PROGRAM Permissives
VAR
	
	
END_VAR

IF (LCP1_IO.Segment[1].ChargeRly_close = TRUE AND 
	LCP1_IO.Segment[2].ChargeRly_close = TRUE AND
	LCP1_IO.Segment[3].ChargeRly_close = TRUE AND 
	LCP2_IO.Segment[4].ChargeRly_close = TRUE AND 
	LCP2_IO.Segment[5].ChargeRly_close = TRUE AND 
	LCP2_IO.Segment[6].ChargeRly_close = TRUE) OR HMI_DB.AllChargeRelayCloseBP = TRUE
	THEN 
		Permissives_DB.AllChargeRelayClosed := TRUE;
	ELSIF 
		LCP1_IO.Segment[1].ChargeRly_close = FALSE AND 
		LCP1_IO.Segment[2].ChargeRly_close = FALSE AND
		LCP1_IO.Segment[3].ChargeRly_close = FALSE AND 
		LCP2_IO.Segment[4].ChargeRly_close = FALSE AND 
		LCP2_IO.Segment[5].ChargeRly_close = FALSE AND 
		LCP2_IO.Segment[6].ChargeRly_close = FALSE
	THEN
		Permissives_DB.AllChargeRelayClosed := FALSE;
END_IF;

IF (LCP1_IO.Segment[1].Module1To3DumpRly_close = FALSE AND 
	LCP1_IO.Segment[2].Module4To6DumpRly_close = FALSE AND
	LCP1_IO.Segment[3].Module7To9DumpRly_close = FALSE AND
	
	LCP2_IO.Segment[4].Module1To3DumpRly_close = FALSE AND 
	LCP2_IO.Segment[5].Module4To6DumpRly_close = FALSE AND
	LCP2_IO.Segment[6].Module7To9DumpRly_close = FALSE) OR HMI_DB.AllDumpRelaysOpenBP = TRUE
	THEN
		Permissives_DB.AllDumpRelayOpen := TRUE;
		ELSIF
			LCP1_IO.Segment[1].Module1To3DumpRly_close = TRUE AND 
			LCP1_IO.Segment[2].Module4To6DumpRly_close = TRUE AND
			LCP1_IO.Segment[3].Module7To9DumpRly_close = TRUE AND
			LCP2_IO.Segment[4].Module1To3DumpRly_close = TRUE AND
			LCP2_IO.Segment[5].Module4To6DumpRly_close = TRUE AND
			LCP2_IO.Segment[6].Module7To9DumpRly_close = TRUE 
		THEN
			Permissives_DB.AllDumpRelayOpen := FALSE;
END_IF;

IF Permissives_DB.AllChargeRelayClosed = TRUE AND 
	Permissives_DB.AllDumpRelayOpen = TRUE AND
	(Permissives_DB.AllVoltMonBoardStatusOK= TRUE OR HMI_DB.AllVoltMonBoardStatusOKBP = TRUE)  //voltmonitor board has missing packets, so this might be sensitive and might need to bypass
	THEN
		Permissives_DB.ReadyToCharge := TRUE;
	ELSE 
		Permissives_DB.ReadyToCharge := FALSE;
END_IF

IF MCP_IO.Charger[1].voltageFeedback <= Permissives_DB.ChargerVThres AND 
	MCP_IO.Charger[2].voltageFeedback <= Permissives_DB.ChargerVThres AND 
	MCP_IO.Charger[3].voltageFeedback <= Permissives_DB.ChargerVThres AND
	MCP_IO.Charger[4].voltageFeedback <= Permissives_DB.ChargerVThres AND
	MCP_IO.Charger[5].voltageFeedback <= Permissives_DB.ChargerVThres AND
	MCP_IO.Charger[6].voltageFeedback <= Permissives_DB.ChargerVThres
	THEN
		Permissives_DB.ChargerVBelowThres := TRUE;
	ELSE
		Permissives_DB.ChargerVBelowThres := FALSE;
END_IF;

IF MCP_IO.Charger[1].HV_isON = FALSE AND 
	MCP_IO.Charger[2].HV_isON = FALSE AND 
	MCP_IO.Charger[3].HV_isON = FALSE AND
	MCP_IO.Charger[4].HV_isON = FALSE AND
	MCP_IO.Charger[5].HV_isON = FALSE AND
	MCP_IO.Charger[6].HV_isON = FALSE 
	THEN
		Permissives_DB.AllChargerHVisOFF := TRUE;
	ELSE 
		Permissives_DB.AllChargerHVisOFF := FALSE;
END_IF

IF MCP_IO.Charger[1].inhibited = TRUE AND
	MCP_IO.Charger[2].inhibited = TRUE AND
	MCP_IO.Charger[3].inhibited = TRUE AND
	MCP_IO.Charger[4].inhibited = TRUE AND
	MCP_IO.Charger[5].inhibited = TRUE AND
	MCP_IO.Charger[6].inhibited = TRUE
	THEN
		Permissives_DB.AllChargerInhibitON	:= TRUE;
	ELSE
		Permissives_DB.AllChargerInhibitON	:= FALSE;
END_IF;

//add volt fb 1 and 2
IF (ABS(LCP1_IO.Segment[1].Module[1].VoltageFeedback[1]) <= Permissives_DB.CapVoltageThres AND
	ABS(LCP1_IO.Segment[1].Module[1].VoltageFeedback[2]) <= Permissives_DB.CapVoltageThres AND
	ABS(LCP1_IO.Segment[1].Module[2].VoltageFeedback[1]) <= Permissives_DB.CapVoltageThres AND
	ABS(LCP1_IO.Segment[1].Module[2].VoltageFeedback[2]) <= Permissives_DB.CapVoltageThres AND
	ABS(LCP1_IO.Segment[1].Module[3].VoltageFeedback[1]) <= Permissives_DB.CapVoltageThres AND
	ABS(LCP1_IO.Segment[1].Module[3].VoltageFeedback[2]) <= Permissives_DB.CapVoltageThres AND
	ABS(LCP1_IO.Segment[2].Module[4].VoltageFeedback[1]) <= Permissives_DB.CapVoltageThres AND
	ABS(LCP1_IO.Segment[2].Module[4].VoltageFeedback[2]) <= Permissives_DB.CapVoltageThres AND
	ABS(LCP1_IO.Segment[2].Module[5].VoltageFeedback[1]) <= Permissives_DB.CapVoltageThres AND
	ABS(LCP1_IO.Segment[2].Module[5].VoltageFeedback[2]) <= Permissives_DB.CapVoltageThres AND
	ABS(LCP1_IO.Segment[2].Module[6].VoltageFeedback[1]) <= Permissives_DB.CapVoltageThres AND
	ABS(LCP1_IO.Segment[2].Module[6].VoltageFeedback[2]) <= Permissives_DB.CapVoltageThres AND
	ABS(LCP1_IO.Segment[3].Module[7].VoltageFeedback[1]) <= Permissives_DB.CapVoltageThres AND
	ABS(LCP1_IO.Segment[3].Module[7].VoltageFeedback[2]) <= Permissives_DB.CapVoltageThres AND
	ABS(LCP1_IO.Segment[3].Module[8].VoltageFeedback[1]) <= Permissives_DB.CapVoltageThres AND 
	ABS(LCP1_IO.Segment[3].Module[8].VoltageFeedback[2]) <= Permissives_DB.CapVoltageThres AND
	ABS(LCP1_IO.Segment[3].Module[9].VoltageFeedback[1]) <= Permissives_DB.CapVoltageThres AND
	ABS(LCP1_IO.Segment[3].Module[9].VoltageFeedback[2]) <= Permissives_DB.CapVoltageThres AND
	
	ABS(LCP2_IO.Segment[4].Module[1].VoltageFeedback[1]) <= Permissives_DB.CapVoltageThres AND
	ABS(LCP2_IO.Segment[4].Module[1].VoltageFeedback[2]) <= Permissives_DB.CapVoltageThres AND
	ABS(LCP2_IO.Segment[4].Module[2].VoltageFeedback[1]) <= Permissives_DB.CapVoltageThres AND
	ABS(LCP2_IO.Segment[4].Module[2].VoltageFeedback[2]) <= Permissives_DB.CapVoltageThres AND
	ABS(LCP2_IO.Segment[4].Module[3].VoltageFeedback[1]) <= Permissives_DB.CapVoltageThres AND
	ABS(LCP2_IO.Segment[4].Module[3].VoltageFeedback[2]) <= Permissives_DB.CapVoltageThres AND
	ABS(LCP2_IO.Segment[5].Module[4].VoltageFeedback[1]) <= Permissives_DB.CapVoltageThres AND
	ABS(LCP2_IO.Segment[5].Module[4].VoltageFeedback[2]) <= Permissives_DB.CapVoltageThres AND
	ABS(LCP2_IO.Segment[5].Module[5].VoltageFeedback[1]) <= Permissives_DB.CapVoltageThres AND
	ABS(LCP2_IO.Segment[5].Module[5].VoltageFeedback[2]) <= Permissives_DB.CapVoltageThres AND
	ABS(LCP2_IO.Segment[5].Module[6].VoltageFeedback[1]) <= Permissives_DB.CapVoltageThres AND
	ABS(LCP2_IO.Segment[5].Module[6].VoltageFeedback[2]) <= Permissives_DB.CapVoltageThres AND
	ABS(LCP2_IO.Segment[6].Module[7].VoltageFeedback[1]) <= Permissives_DB.CapVoltageThres AND
	ABS(LCP2_IO.Segment[6].Module[7].VoltageFeedback[2]) <= Permissives_DB.CapVoltageThres AND
	ABS(LCP2_IO.Segment[6].Module[8].VoltageFeedback[1]) <= Permissives_DB.CapVoltageThres AND 
	ABS(LCP2_IO.Segment[6].Module[8].VoltageFeedback[2]) <= Permissives_DB.CapVoltageThres AND
	ABS(LCP2_IO.Segment[6].Module[9].VoltageFeedback[1]) <= Permissives_DB.CapVoltageThres AND
	ABS(LCP2_IO.Segment[6].Module[9].VoltageFeedback[2]) <= Permissives_DB.CapVoltageThres) OR HMI_DB.AllCapsDischargedBP = TRUE 
(*  AND all other module voltage feedback <= 40, might need the -ve end & check for valid data*) 
	THEN
		Permissives_DB.AllCapsDischarged := TRUE;
	ELSE 
		Permissives_DB.AllCapsDischarged := FALSE;
END_IF

//VTB status
//LCP1 Voltage Monitor Board bat lo
IF LCP1_IO.VMB.VTB[0].BateryLow = TRUE OR 
	LCP1_IO.VMB.VTB[1].BateryLow = TRUE OR 
	LCP1_IO.VMB.VTB[2].BateryLow = TRUE OR 
	LCP1_IO.VMB.VTB[3].BateryLow = TRUE OR 
	LCP1_IO.VMB.VTB[4].BateryLow = TRUE OR 
	LCP1_IO.VMB.VTB[5].BateryLow = TRUE OR 
	LCP1_IO.VMB.VTB[6].BateryLow = TRUE OR 
	LCP1_IO.VMB.VTB[7].BateryLow = TRUE OR 
	LCP1_IO.VMB.VTB[8].BateryLow = TRUE OR 
	LCP1_IO.VMB.VTB[9].BateryLow = TRUE OR 
	LCP1_IO.VMB.VTB[10].BateryLow = TRUE OR 
	LCP1_IO.VMB.VTB[11].BateryLow = TRUE OR 
	LCP1_IO.VMB.VTB[12].BateryLow = TRUE OR 
	LCP1_IO.VMB.VTB[13].BateryLow = TRUE OR 
	LCP1_IO.VMB.VTB[14].BateryLow = TRUE OR 
	LCP1_IO.VMB.VTB[15].BateryLow = TRUE OR 
	LCP1_IO.VMB.VTB[16].BateryLow = TRUE OR 
	LCP1_IO.VMB.VTB[17].BateryLow = TRUE 
	THEN 
		Permissives_DB.AnyLCP1MonBoardBatLo := TRUE;
	ELSIF 
		LCP1_IO.VMB.VTB[0].BateryLow = FALSE AND 
		LCP1_IO.VMB.VTB[1].BateryLow = FALSE AND 
		LCP1_IO.VMB.VTB[2].BateryLow = FALSE AND 	
		LCP1_IO.VMB.VTB[3].BateryLow = FALSE AND 
		LCP1_IO.VMB.VTB[4].BateryLow = FALSE AND 
		LCP1_IO.VMB.VTB[5].BateryLow = FALSE AND 
		LCP1_IO.VMB.VTB[6].BateryLow = FALSE AND 
		LCP1_IO.VMB.VTB[7].BateryLow = FALSE AND 
		LCP1_IO.VMB.VTB[8].BateryLow = FALSE AND 
		LCP1_IO.VMB.VTB[9].BateryLow = FALSE AND 
		LCP1_IO.VMB.VTB[10].BateryLow = FALSE AND 
		LCP1_IO.VMB.VTB[11].BateryLow = FALSE AND 
		LCP1_IO.VMB.VTB[12].BateryLow = FALSE AND 
		LCP1_IO.VMB.VTB[13].BateryLow = FALSE AND 
		LCP1_IO.VMB.VTB[14].BateryLow = FALSE AND 
		LCP1_IO.VMB.VTB[15].BateryLow = FALSE AND 
		LCP1_IO.VMB.VTB[16].BateryLow = FALSE AND 
		LCP1_IO.VMB.VTB[17].BateryLow = FALSE 
	THEN 
		Permissives_DB.AnyLCP1MonBoardBatLo := FALSE;
END_IF	
//LCP2 Voltage Monitor Board battery lo
IF LCP2_IO.VMB.VTB[0].BateryLow = TRUE OR 
	LCP2_IO.VMB.VTB[1].BateryLow = TRUE OR 
	LCP2_IO.VMB.VTB[2].BateryLow = TRUE OR 
	LCP2_IO.VMB.VTB[3].BateryLow = TRUE OR 
	LCP2_IO.VMB.VTB[4].BateryLow = TRUE OR 
	LCP2_IO.VMB.VTB[5].BateryLow = TRUE OR 
	LCP2_IO.VMB.VTB[6].BateryLow = TRUE OR 
	LCP2_IO.VMB.VTB[7].BateryLow = TRUE OR 
	LCP2_IO.VMB.VTB[8].BateryLow = TRUE OR 
	LCP2_IO.VMB.VTB[9].BateryLow = TRUE OR 
	LCP2_IO.VMB.VTB[10].BateryLow = TRUE OR 
	LCP2_IO.VMB.VTB[11].BateryLow = TRUE OR 
	LCP2_IO.VMB.VTB[12].BateryLow = TRUE OR 
	LCP2_IO.VMB.VTB[13].BateryLow = TRUE OR 
	LCP2_IO.VMB.VTB[14].BateryLow = TRUE OR 
	LCP2_IO.VMB.VTB[15].BateryLow = TRUE OR 
	LCP2_IO.VMB.VTB[16].BateryLow = TRUE OR 
	LCP2_IO.VMB.VTB[17].BateryLow = TRUE 
	THEN 
		Permissives_DB.AnyLCP2MonBoardBatLo := TRUE;
	ELSIF 
		LCP2_IO.VMB.VTB[0].BateryLow = FALSE AND 
		LCP2_IO.VMB.VTB[1].BateryLow = FALSE AND 
		LCP2_IO.VMB.VTB[2].BateryLow = FALSE AND 	
		LCP2_IO.VMB.VTB[3].BateryLow = FALSE AND 
		LCP2_IO.VMB.VTB[4].BateryLow = FALSE AND 
		LCP2_IO.VMB.VTB[5].BateryLow = FALSE AND 
		LCP2_IO.VMB.VTB[6].BateryLow = FALSE AND 
		LCP2_IO.VMB.VTB[7].BateryLow = FALSE AND 
		LCP2_IO.VMB.VTB[8].BateryLow = FALSE AND 
		LCP2_IO.VMB.VTB[9].BateryLow = FALSE AND 
		LCP2_IO.VMB.VTB[10].BateryLow = FALSE AND 
		LCP2_IO.VMB.VTB[11].BateryLow = FALSE AND 
		LCP2_IO.VMB.VTB[12].BateryLow = FALSE AND 
		LCP2_IO.VMB.VTB[13].BateryLow = FALSE AND 
		LCP2_IO.VMB.VTB[14].BateryLow = FALSE AND 
		LCP2_IO.VMB.VTB[15].BateryLow = FALSE AND 
		LCP2_IO.VMB.VTB[16].BateryLow = FALSE AND 
		LCP2_IO.VMB.VTB[17].BateryLow = FALSE 
	THEN 
		Permissives_DB.AnyLCP2MonBoardBatLo := FALSE;
END_IF	
//lcp1 volt montiro board loss HB
IF LCP1_IO.VMB.VTB[0].LossVoltTransBoard = TRUE OR 
	LCP1_IO.VMB.VTB[1].LossVoltTransBoard = TRUE OR 
	LCP1_IO.VMB.VTB[2].LossVoltTransBoard = TRUE OR 
	LCP1_IO.VMB.VTB[3].LossVoltTransBoard = TRUE OR 
	LCP1_IO.VMB.VTB[4].LossVoltTransBoard = TRUE OR 
	LCP1_IO.VMB.VTB[5].LossVoltTransBoard = TRUE OR 
	LCP1_IO.VMB.VTB[6].LossVoltTransBoard = TRUE OR 
	LCP1_IO.VMB.VTB[7].LossVoltTransBoard = TRUE OR 
	LCP1_IO.VMB.VTB[8].LossVoltTransBoard = TRUE OR 
	LCP1_IO.VMB.VTB[9].LossVoltTransBoard = TRUE OR 
	LCP1_IO.VMB.VTB[10].LossVoltTransBoard = TRUE OR 
	LCP1_IO.VMB.VTB[11].LossVoltTransBoard = TRUE OR 
	LCP1_IO.VMB.VTB[12].LossVoltTransBoard = TRUE OR 
	LCP1_IO.VMB.VTB[13].LossVoltTransBoard = TRUE OR 
	LCP1_IO.VMB.VTB[14].LossVoltTransBoard = TRUE OR 
	LCP1_IO.VMB.VTB[15].LossVoltTransBoard = TRUE OR 
	LCP1_IO.VMB.VTB[16].LossVoltTransBoard = TRUE OR 
	LCP1_IO.VMB.VTB[17].LossVoltTransBoard = TRUE 
	THEN 
		Permissives_DB.AnyLCP1MonBoardLoss := TRUE;
	ELSIF 
		LCP1_IO.VMB.VTB[0].LossVoltTransBoard = FALSE AND 
		LCP1_IO.VMB.VTB[1].LossVoltTransBoard = FALSE AND 
		LCP1_IO.VMB.VTB[2].LossVoltTransBoard = FALSE AND 	
		LCP1_IO.VMB.VTB[3].LossVoltTransBoard = FALSE AND 
		LCP1_IO.VMB.VTB[4].LossVoltTransBoard = FALSE AND 
		LCP1_IO.VMB.VTB[5].LossVoltTransBoard = FALSE AND 
		LCP1_IO.VMB.VTB[6].LossVoltTransBoard = FALSE AND 
		LCP1_IO.VMB.VTB[7].LossVoltTransBoard = FALSE AND 
		LCP1_IO.VMB.VTB[8].LossVoltTransBoard = FALSE AND 
		LCP1_IO.VMB.VTB[9].LossVoltTransBoard = FALSE AND 
		LCP1_IO.VMB.VTB[10].LossVoltTransBoard = FALSE AND 
		LCP1_IO.VMB.VTB[11].LossVoltTransBoard = FALSE AND 
		LCP1_IO.VMB.VTB[12].LossVoltTransBoard = FALSE AND 
		LCP1_IO.VMB.VTB[13].LossVoltTransBoard = FALSE AND 
		LCP1_IO.VMB.VTB[14].LossVoltTransBoard = FALSE AND 
		LCP1_IO.VMB.VTB[15].LossVoltTransBoard = FALSE AND 
		LCP1_IO.VMB.VTB[16].LossVoltTransBoard = FALSE AND 
		LCP1_IO.VMB.VTB[17].LossVoltTransBoard = FALSE 
	THEN 
		Permissives_DB.AnyLCP1MonBoardLoss := FALSE;
END_IF 
//lcp2 volt montiro board loss HB
IF LCP2_IO.VMB.VTB[0].LossVoltTransBoard = TRUE OR 
	LCP2_IO.VMB.VTB[1].LossVoltTransBoard = TRUE OR 
	LCP2_IO.VMB.VTB[2].LossVoltTransBoard = TRUE OR 
	LCP2_IO.VMB.VTB[3].LossVoltTransBoard = TRUE OR 
	LCP2_IO.VMB.VTB[4].LossVoltTransBoard = TRUE OR 
	LCP2_IO.VMB.VTB[5].LossVoltTransBoard = TRUE OR 
	LCP2_IO.VMB.VTB[6].LossVoltTransBoard = TRUE OR 
	LCP2_IO.VMB.VTB[7].LossVoltTransBoard = TRUE OR 
	LCP2_IO.VMB.VTB[8].LossVoltTransBoard = TRUE OR 
	LCP2_IO.VMB.VTB[9].LossVoltTransBoard = TRUE OR 
	LCP2_IO.VMB.VTB[10].LossVoltTransBoard = TRUE OR 
	LCP2_IO.VMB.VTB[11].LossVoltTransBoard = TRUE OR 
	LCP2_IO.VMB.VTB[12].LossVoltTransBoard = TRUE OR 
	LCP2_IO.VMB.VTB[13].LossVoltTransBoard = TRUE OR 
	LCP2_IO.VMB.VTB[14].LossVoltTransBoard = TRUE OR 
	LCP2_IO.VMB.VTB[15].LossVoltTransBoard = TRUE OR 
	LCP2_IO.VMB.VTB[16].LossVoltTransBoard = TRUE OR 
	LCP2_IO.VMB.VTB[17].LossVoltTransBoard = TRUE 
	THEN 
		Permissives_DB.AnyLCP2MonBoardLoss := TRUE;
	ELSIF 
		LCP2_IO.VMB.VTB[0].LossVoltTransBoard = FALSE AND 
		LCP2_IO.VMB.VTB[1].LossVoltTransBoard = FALSE AND 
		LCP2_IO.VMB.VTB[2].LossVoltTransBoard = FALSE AND 	
		LCP2_IO.VMB.VTB[3].LossVoltTransBoard = FALSE AND 
		LCP2_IO.VMB.VTB[4].LossVoltTransBoard = FALSE AND 
		LCP2_IO.VMB.VTB[5].LossVoltTransBoard = FALSE AND 
		LCP2_IO.VMB.VTB[6].LossVoltTransBoard = FALSE AND 
		LCP2_IO.VMB.VTB[7].LossVoltTransBoard = FALSE AND 
		LCP2_IO.VMB.VTB[8].LossVoltTransBoard = FALSE AND 
		LCP2_IO.VMB.VTB[9].LossVoltTransBoard = FALSE AND 
		LCP2_IO.VMB.VTB[10].LossVoltTransBoard = FALSE AND 
		LCP2_IO.VMB.VTB[11].LossVoltTransBoard = FALSE AND 
		LCP2_IO.VMB.VTB[12].LossVoltTransBoard = FALSE AND 
		LCP2_IO.VMB.VTB[13].LossVoltTransBoard = FALSE AND 
		LCP2_IO.VMB.VTB[14].LossVoltTransBoard = FALSE AND 
		LCP2_IO.VMB.VTB[15].LossVoltTransBoard = FALSE AND 
		LCP2_IO.VMB.VTB[16].LossVoltTransBoard = FALSE AND 
		LCP2_IO.VMB.VTB[17].LossVoltTransBoard = FALSE 
	THEN 
		Permissives_DB.AnyLCP2MonBoardLoss := FALSE;
END_IF 

IF Permissives_DB.AnyLCP1MonBoardBatLo = TRUE OR Permissives_DB.AnyLCP2MonBoardBatLo = TRUE 
	THEN 
		Permissives_DB.AnyVoltMonBoardBatLo := TRUE;
	ELSIF 
		Permissives_DB.AnyLCP1MonBoardBatLo = FALSE AND Permissives_DB.AnyLCP2MonBoardBatLo = FALSE 
	THEN 
		Permissives_DB.AnyVoltMonBoardBatLo := FALSE;
END_IF

IF Permissives_DB.AnyLCP1MonBoardLoss = TRUE OR Permissives_DB.AnyLCP2MonBoardLoss = TRUE 
	THEN 
		Permissives_DB.AnyVoltMonBoardLoss := TRUE;
	ELSIF 
		Permissives_DB.AnyLCP1MonBoardLoss = FALSE AND Permissives_DB.AnyLCP2MonBoardLoss = FALSE 
	THEN 
		Permissives_DB.AnyVoltMonBoardLoss := FALSE;
END_IF

IF (Permissives_DB.ChargerVBelowThres = TRUE AND 
	Permissives_DB.AllChargerHVisOFF = TRUE AND 
	//Permissives_DB.AllChargerInhibitON	= TRUE AND 
	Permissives_DB.AllDumpRelayOpen = FALSE AND 
	Permissives_DB.AllCapsDischarged = TRUE) OR HMI_DB.SystemSafeBP = TRUE 
THEN
	(*MCP_IO.Charger[2].voltageFeedback <= 10 AND *)
	Permissives_DB.SystemIsSafe := TRUE;
	ELSE
		Permissives_DB.SystemIsSafe := FALSE;
END_IF
		
IF Permissives_DB.AllCapsDischarged = TRUE THEN 
	LCP1_IO.SegmentCharged := FALSE; //for status light only
	LCP2_IO.SegmentCharged := FALSE; //for status light only
END_IF

IF MCP_IO.Charger[1].EndOfCharge = TRUE AND
	MCP_IO.Charger[2].EndOfCharge = TRUE AND
	MCP_IO.Charger[3].EndOfCharge = TRUE AND
	MCP_IO.Charger[4].EndOfCharge = TRUE AND
	MCP_IO.Charger[5].EndOfCharge = TRUE AND
	MCP_IO.Charger[6].EndOfCharge = TRUE 
THEN
	Permissives_DB.AllChargerEOC := TRUE;
	ELSE
		Permissives_DB.AllChargerEOC := FALSE;
END_IF;

// might or might not beused for the seq
IF MCP_IO.PSU1_DCOK = TRUE AND LCP1_IO.PSU1OK = TRUE AND LCP2_IO.PSU1OK = TRUE THEN
	Trips_DB.AllDCpsuOK := TRUE;
	ELSE
		Trips_DB.AllDCpsuOK := FALSE;
END_IF

IF MCP_IO.MasterStopPB_NotPressed = FALSE THEN 
	Trips_DB.MasterSTOPPressed := TRUE;
	ELSE
		Trips_DB.MasterSTOPPressed := FALSE;
END_IF

IF MCP_IO.CageEstopCircuitOK = FALSE OR MCP_IO.MasterStopPB_NotPressed = FALSE THEN 
	Trips_DB.AnyEstopPressed := TRUE;
END_IF

END_PROGRAM

(* stored: Version 1.1.0.1, ProductVersion 3.1.4024.11
   POU Permissives: Id {639d0291-603e-4994-93d7-3ec14345fa0c}, SpecialFunc None *)
